// TIA Portal V21 program export: 0 tag tables, 0 data types, 2 data blocks, 2 code blocks (in call order from the OBs), 0 instance data blocks

DATA_BLOCK "Data_block_1"   // DB1
{ S7_Optimized_Access := 'TRUE' }
// stored: MemoryReserve 100
   VAR
      Variable1 : Bool;
      Variable2 : Int := 16;
   END_VAR
BEGIN
END_DATA_BLOCK

DATA_BLOCK "Data_block_11"   // DB2
{ S7_Optimized_Access := 'TRUE' }
// stored: MemoryReserve 100
   VAR
      var1 : Bool;
   END_VAR
BEGIN
END_DATA_BLOCK

ORGANIZATION_BLOCK "Main"   // OB1, LAD, ProgramCycle
TITLE = "Main Program Sweep (Cycle)"
{ S7_Optimized_Access := 'TRUE' }
// stored: SetENOAutomatically false
   VAR_INPUT
      Initial_Call : Bool;   // Initial call of this OB
      Remanence : Bool;   // =True, if remanent data are available
   END_VAR
BEGIN
END_ORGANIZATION_BLOCK

ORGANIZATION_BLOCK "CyclicInterrupt"
{ S7_Optimized_Access := 'TRUE' }
VERSION: 0.1

BEGIN
IF THIS THEN
	that := TRUE;
END_IF;

END_ORGANIZATION_BLOCK
